FUNCTION_BLOCK ConfirmationButton
  (* Standard: 61499-2 *)
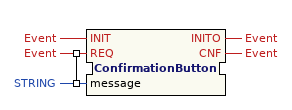
  EVENT_INPUT
    INIT;
    REQ WITH message;
  END_EVENT
  EVENT_OUTPUT
    INITO;
    CNF;
  END_EVENT
  VAR_INPUT
    message : STRING;
  END_VAR
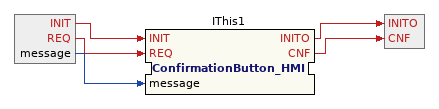
  FBS
    IThis1 : ConfirmationButton_HMI;
  END_FBS
  EVENT_CONNECTIONS
    INIT TO IThis1.INIT;
    REQ TO IThis1.REQ;
    IThis1.INITO TO INITO;
    IThis1.CNF TO CNF;
  END_CONNECTIONS
  DATA_CONNECTIONS
    message TO IThis1.message;
  END_CONNECTIONS
END_FUNCTION_BLOCK
